// TwinCAT 3 PLC project Untitled1
// ProgramVersion: 3.1.4023.0
// libraries:
//   Tc2_HVAC, * (Beckhoff Automation GmbH)
//   Tc2_Standard, * (Beckhoff Automation GmbH)
//   Tc2_System, * (Beckhoff Automation GmbH)
//   Tc3_Module, * (Beckhoff Automation GmbH)
// project tree:
//   / PlcTask.TcTTO
//   POUs/ BARFanCoil.TcPOU, MAIN.TcPOU
//   POUs/HVAC/ AnalogInput.TcPOU, AnalogOutputEx.TcPOU, AntiBlockingDamper.TcPOU, AntiBlockingPump.TcPOU, CirculationPumpEx.TcPOU, Motor1Speed.TcPOU, Motor2Speed.TcPOU, Motor3Speed.TcPOU (not stored), OverwriteAnalog.TcPOU (not stored), Scheduler28ch.TcPOU, Scheduler7ch.TcPOU, SchedulerPublicHolidays.TcPOU, SchedulerSpecialPeriods.TcPOU (not stored), TemperatureSensorEx2.TcPOU (not stored), ThreePointActuatorMode.TcPOU, TwoPointActuatorMode.TcPOU (not stored), Work.TcPOU (not stored)
// real-time tasks:
//   TASK PlcTask: cycle T#10ms, priority 20, ADS port 350

CONFIGURATION Untitled1
    RESOURCE PLC ON TwinCAT3
        TASK PlcTask(INTERVAL := T#10ms, PRIORITY := 20);
        PROGRAM MAIN WITH PlcTask : MAIN;
    END_RESOURCE
END_CONFIGURATION

// ---- POUs/MAIN.TcPOU
PROGRAM MAIN
VAR
	
END_VAR

CirculationPumpEx();
AntiBlockingPump();
Work();
Scheduler7ch();
Scheduler28ch();
SchedulerSpecialPeriods();
SchedulerPublicHolidays();
Motor1Speed();
Motor2Speed();
Motor3Speed();
TwoPointActuatorMode();
ThreePointActuatorMode();
TemperatureSensorEx2();
OverwriteAnalog();
AnalogInput();
AnalogOutputEx();
AntiBlockingDamper();
BARFanCoil();

END_PROGRAM

// ---- POUs/HVAC/CirculationPumpEx.TcPOU
PROGRAM CirculationPumpEx
VAR
	fbHVACCirculationPumpEx: FB_HVACCirculationPumpEx;
	eDataSecurityType: E_HVACDataSecurityType := E_HVACDataSecurityType.eHVACDataSecurityType_Idle;
	bSetDefault: BOOL;
	bEnable: BOOL := TRUE;
	bExternal: BOOL;
	eCtrlModeActuator: E_HVACActuatorMode;
	rOutsideTemp: REAL;
	rValvePosition: REAL;
	bFeedbPump: BOOL := TRUE;
	bPumpProtec: BOOL := TRUE;
	bManSwitch: BOOL := TRUE;
	bCtrlVoltage: BOOL := TRUE;
	bReset: BOOL;
	bPump: BOOL;
	byState: BYTE;
	bReqExternal: BOOL;
	bReqOutsideTemp: BOOL;
	bReqValve: BOOL;
	bStateManSwitch: BOOL;
	udiSecRT_StopDelay: UDINT;
	udiSecRT_FeedbPumpDelay: UDINT;
	eStateModeActuator: Tc2_HVAC.E_HVACActuatorMode;
	bError: BOOL;
	byError: BYTE;
	bErrorPumpProtec: BOOL;
	bErrorFeedb: BOOL;
	bInvalidParameter: BOOL;
	udiSecStopDelay: UDINT;
	udiSecFeedbPumpDelay: UDINT;
	rOutsideTempHighLimit: REAL;
	rOutsideTempLowLimit: REAL;
	rValvePositionLimitOn: REAL;
	rValvePositionLimitOff: REAL;
	eReqPump: E_HVACReqPump;
END_VAR

fbHVACCirculationPumpEx(
	eDataSecurityType:=eDataSecurityType, 
	bSetDefault:=bSetDefault, 
	bEnable:=bEnable, 
	bExternal:=bExternal, 
	eCtrlModeActuator:=eCtrlModeActuator, 
	rOutsideTemp:=rOutsideTemp, 
	rValvePosition:=rValvePosition, 
	bFeedbPump:=bFeedbPump, 
	bPumpProtec:=bPumpProtec, 
	bManSwitch:=bManSwitch, 
	bCtrlVoltage:=bCtrlVoltage, 
	bReset:=bReset, 
	bPump=>bPump, 
	byState=>byState, 
	bReqExternal=>bReqExternal, 
	bReqOutsideTemp=>bReqOutsideTemp, 
	bReqValve=>bReqValve, 
	bStateManSwitch=>bStateManSwitch, 
	udiSecRT_StopDelay=>udiSecRT_StopDelay, 
	udiSecRT_FeedbPumpDelay=>udiSecRT_FeedbPumpDelay, 
	eStateModeActuator=>eStateModeActuator, 
	bError=>bError, 
	byError=>byError, 
	bErrorPumpProtec=>bErrorPumpProtec, 
	bErrorFeedb=>bErrorFeedb, 
	bInvalidParameter=>bInvalidParameter, 
	udiSecStopDelay:=udiSecStopDelay, 
	udiSecFeedbPumpDelay:=udiSecFeedbPumpDelay, 
	rOutsideTempHighLimit:=rOutsideTempHighLimit, 
	rOutsideTempLowLimit:=rOutsideTempLowLimit, 
	rValvePositionLimitOn:=rValvePositionLimitOn, 
	rValvePositionLimitOff:=rValvePositionLimitOff, 
	eReqPump:=eReqPump);

END_PROGRAM

// ---- POUs/HVAC/AntiBlockingPump.TcPOU
PROGRAM AntiBlockingPump
VAR
	fbHVACAntiBlockingPump: FB_HVACAntiBlockingPump;
	eDataSecurityType: E_HVACDataSecurityType := E_HVACDataSecurityType.eHVACDataSecurityType_Idle;
	bSetDefault: BOOL;
	bEnable: BOOL;
	bDisable: BOOL;
	bIn: BOOL;
	dtSystemTime: DATE_AND_TIME;
	bReset: BOOL;
	eAntiBlockingMode: E_HVACAntiBlockingMode;
	iHoursDowntime: INT;
	iDayWeekly: INT;
	iHour: INT;
	iMinute: INT;
	iLenghtImpulse: INT;
	bOut: BOOL;
	bOutAndAntiBlocking: BOOL;
	bQAntiBlocking: BOOL;
	bInvalidParameter: BOOL;
END_VAR

fbHVACAntiBlockingPump(
	eDataSecurityType:=eDataSecurityType, 
	bSetDefault:=bSetDefault, 
	bEnable:=bEnable, 
	bDisable:=bDisable, 
	bIn:=bIn, 
	dtSystemTime:=dtSystemTime, 
	bReset:=bReset, 
	eAntiBlockingMode:=eAntiBlockingMode, 
	iHoursDowntime:=iHoursDowntime, 
	iDayWeekly:=iDayWeekly, 
	iHour:=iHour, 
	iMinute:=iMinute, 
	iLenghtImpulse:=iLenghtImpulse, 
	bOut=>bOut, 
	bOutAndAntiBlocking=>bOutAndAntiBlocking, 
	bQAntiBlocking=>bQAntiBlocking, 
	bInvalidParameter=>bInvalidParameter);

END_PROGRAM

// ---- POUs/HVAC/Scheduler7ch.TcPOU
PROGRAM Scheduler7ch
VAR
	fbHVACScheduler7ch:FB_HVACScheduler7ch;
	eDataSecurityType:E_HVACDataSecurityType := E_HVACDataSecurityType.eHVACDataSecurityType_Idle;
	bSetDefault:BOOL;
	bEnable:BOOL;
	dtSystemTime:DT;
	uiOffsetBefore:UINT;
	bReset:BOOL;
	arrTimeChannel:ARRAY[1..7] OF ST_HVACTimeChannel;
	bOutput:BOOL;
	bEdgeOn:BOOL;
	bEdgeOff:BOOL;
	tNextOn:TIME;
	tNextOff:TIME;
	bInvalidParameter:BOOL;
END_VAR

fbHVACScheduler7ch(
	eDataSecurityType:=eDataSecurityType , 
	bSetDefault:=bSetDefault, 
	bEnable:=bEnable , 
	dtSystemTime:=dtSystemTime , 
	uiOffsetBefore:=uiOffsetBefore, 
	bReset:=bReset, 
	arrTimeChannel:=arrTimeChannel, 
	bOutput=>bOutput, 
	bEdgeOn=>bEdgeOn, 
	bEdgeOff=>bEdgeOff, 
	tNextOn=>tNextOn, 
	tNextOff=>tNextOff, 
	bInvalidParameter=>bInvalidParameter
);

END_PROGRAM

// ---- POUs/HVAC/Scheduler28ch.TcPOU
PROGRAM Scheduler28ch
VAR
	fbHVACScheduler28ch:FB_HVACScheduler28ch;
	eDataSecurityType:E_HVACDataSecurityType := E_HVACDataSecurityType.eHVACDataSecurityType_Idle;
	bSetDefault:BOOL;
	bEnable:BOOL;
	dtSystemTime:DT;
	uiOffsetBefore:UINT;
	bReset:BOOL;
	arrTimeChannel2:ARRAY[1..28] OF ST_HVACTimeChannel;
	bOutput:BOOL;
	bEdgeOn:BOOL;
	bEdgeOff:BOOL;
	tNextOn:TIME;
	tNextOff:TIME;
	bInvalidParameter:BOOL;
END_VAR

fbHVACScheduler28ch(
	eDataSecurityType:=eDataSecurityType , 
	bSetDefault:=bSetDefault, 
	bEnable:=bEnable , 
	dtSystemTime:=dtSystemTime , 
	uiOffsetBefore:=uiOffsetBefore, 
	bReset:=bReset, 
	arrTimeChannel:=arrTimeChannel2, 
	bOutput=>bOutput, 
	bEdgeOn=>bEdgeOn, 
	bEdgeOff=>bEdgeOff, 
	tNextOn=>tNextOn, 
	tNextOff=>tNextOff, 
	bInvalidParameter=>bInvalidParameter
);

END_PROGRAM

// ---- POUs/HVAC/SchedulerPublicHolidays.TcPOU
PROGRAM SchedulerPublicHolidays
VAR
	fbHVACSchedulerPublicHolidays:FB_HVACSchedulerPublicHolidays;
	eDataSecurityType:E_HVACDataSecurityType := E_HVACDataSecurityType.eHVACDataSecurityType_Idle;
	bSetDefault:BOOL;
	bEnable:BOOL;
	dtSystemTime:DT;
	bReset:BOOL;
	arrHoliday:ARRAY[1..20] OF ST_HVACHoliday;
	bOutput:BOOL;
	bEdgeOn:BOOL;
	bEdgeOff:BOOL;
	tNextOn:TIME;
	tNextOff:TIME;
	bInvalidParameter:BOOL;
END_VAR

fbHVACSchedulerPublicHolidays(
	eDataSecurityType:=eDataSecurityType , 
	bSetDefault:= bSetDefault, 
	bEnable:=bEnable, 
	dtSystemTime:=dtSystemTime, 
	bReset:=bReset, 
	arrHoliday:=arrHoliday, 
	bOutput=>bOutput, 
	bEdgeOn=>bEdgeOn, 
	bEdgeOff=>bEdgeOff, 
	tNextOn=>tNextOn, 
	tNextOff=>tNextOff, 
	bInvalidParameter=>bInvalidParameter);

END_PROGRAM

// ---- POUs/HVAC/Motor1Speed.TcPOU
PROGRAM Motor1Speed
VAR
	fbHVACMotor1Speed: FB_HVACMotor1Speed;
	eDataSecurityType: E_HVACDataSecurityType := E_HVACDataSecurityType.eHVACDataSecurityType_Idle;
	bSetDefault: BOOL;
	bEnable: BOOL;
	bAuto: BOOL;
	eCtrlModeActuator: E_HVACActuatorMode;
	bMotorProtec: BOOL;
	bFeedbContactor: BOOL;
	bFeedbProcess: BOOL;
	bRepairSwitch: BOOL;
	bManSwitch: BOOL;
	bCtrlVoltage: BOOL;
	bReset: BOOL;
	bMotor: BOOL;
	byState: BYTE;
	bStateAuto: BOOL;
	bStateRepairSwitch: BOOL;
	bStateManSwitch: BOOL;
	eStateModeActuator: Tc2_HVAC.E_HVACActuatorMode;
	bErrorGeneral: BOOL;
	byError: BYTE;
	bErrorMotorprotec: BOOL;
	bErrorFeedbContactor: BOOL;
	bErrorFeedbProcess: BOOL;
	bInvalidParameter: BOOL;
	tStartDelay: TIME;
	tStopDelay: TIME;
	tDelayFeedbContactor: TIME;
	tFeedbProcessTimer: TIME;
	tDelayFeedbProcess: TIME;
END_VAR

fbHVACMotor1Speed(
	eDataSecurityType:=eDataSecurityType, 
	bSetDefault:=bSetDefault, 
	bEnable:=bEnable, 
	bAuto:=bAuto, 
	eCtrlModeActuator:=eCtrlModeActuator, 
	bMotorProtec:=bMotorProtec, 
	bFeedbContactor:=bFeedbContactor, 
	bFeedbProcess:=bFeedbProcess, 
	bRepairSwitch:=bRepairSwitch, 
	bManSwitch:=bManSwitch, 
	bCtrlVoltage:=bCtrlVoltage, 
	bReset:=bReset, 
	bMotor=>bMotor, 
	byState=>byState, 
	bStateAuto=>bStateAuto, 
	bStateRepairSwitch=>bStateRepairSwitch, 
	bStateManSwitch=>bStateManSwitch, 
	eStateModeActuator=>eStateModeActuator, 
	bErrorGeneral=>bErrorGeneral, 
	byError=>byError, 
	bErrorMotorprotec=>bErrorMotorprotec, 
	bErrorFeedbContactor=>bErrorFeedbContactor, 
	bErrorFeedbProcess=>bErrorFeedbProcess, 
	bInvalidParameter=>bInvalidParameter, 
	tStartDelay:=tStartDelay, 
	tStopDelay:=tStopDelay, 
	tDelayFeedbContactor:=tDelayFeedbContactor, 
	tFeedbProcessTimer:=tFeedbProcessTimer, 
	tDelayFeedbProcess:=tDelayFeedbProcess);

END_PROGRAM

// ---- POUs/HVAC/Motor2Speed.TcPOU
PROGRAM Motor2Speed
VAR
	fbHVACMotor2Speed: FB_HVACMotor2Speed;
	eDataSecurityType: E_HVACDataSecurityType := E_HVACDataSecurityType.eHVACDataSecurityType_Idle;
	bSetDefault: BOOL;
	bEnable: BOOL;
	bAutoSpeed1: BOOL;
	bAutoSpeed2: BOOL;
	eCtrlModeActuator: E_HVACActuatorMode;
	bMotorProtecSpeed1: BOOL;
	bMotorProtecSpeed2: BOOL;
	bFeedbContactorSpeed1: BOOL;
	bFeedbContactorSpeed2: BOOL;
	bFeedbProcess: BOOL;
	bRepairSwitch: BOOL;
	bManSwitch: BOOL;
	bCtrlVoltage: BOOL;
	bReset: BOOL;
	bMotorSpeed1: BOOL;
	bMotorSpeed2: BOOL;
	byState: BYTE;
	bStateAutoSpeed1: BOOL;
	bStateAutoSpeed2: BOOL;
	bStateRepairSwitch: BOOL;
	bStateManSwitch: BOOL;
	eStateModeActuator: Tc2_HVAC.E_HVACActuatorMode;
	bErrorGeneral: BOOL;
	byError: BYTE;
	bErrorMotorprotecSpeed1: BOOL;
	bErrorMotorprotecSpeed2: BOOL;
	bErrorFeedbContactorSpeed1: BOOL;
	bErrorFeedbContactorSpeed2: BOOL;
	bErrorFeedbProcess: BOOL;
	bInvalidParameter: BOOL;
	tStartDelay: TIME;
	tStopDelay: TIME;
	tDelayFeedbContactorSpeed1: TIME;
	tDelayFeedbContactorSpeed2: TIME;
	tFeedbProcessTimer: TIME;
	tDelayFeedbProcess: TIME;
	tDelaySpeed1: TIME;
	tDelaySpeed1ToSpeed2: TIME;
	tDelaySpeed2ToSpeed1: TIME;
END_VAR

fbHVACMotor2Speed(
	eDataSecurityType:=eDataSecurityType, 
	bSetDefault:=bSetDefault, 
	bEnable:=bEnable, 
	bAutoSpeed1:=bAutoSpeed1, 
	bAutoSpeed2:=bAutoSpeed2, 
	eCtrlModeActuator:=eCtrlModeActuator, 
	bMotorProtecSpeed1:=bMotorProtecSpeed1, 
	bMotorProtecSpeed2:=bMotorProtecSpeed2, 
	bFeedbContactorSpeed1:=bFeedbContactorSpeed1, 
	bFeedbContactorSpeed2:=bFeedbContactorSpeed2, 
	bFeedbProcess:=bFeedbProcess, 
	bRepairSwitch:=bRepairSwitch, 
	bManSwitch:=bManSwitch, 
	bCtrlVoltage:=bCtrlVoltage, 
	bReset:=bReset, 
	bMotorSpeed1=>bMotorSpeed1, 
	bMotorSpeed2=>bMotorSpeed2, 
	byState=>byState, 
	bStateAutoSpeed1=>bStateAutoSpeed1, 
	bStateAutoSpeed2=>bStateAutoSpeed2, 
	bStateRepairSwitch=>bStateRepairSwitch, 
	bStateManSwitch=>bStateManSwitch, 
	eStateModeActuator=>eStateModeActuator, 
	bErrorGeneral=>bErrorGeneral, 
	byError=>byError, 
	bErrorMotorprotecSpeed1=>bErrorMotorprotecSpeed1, 
	bErrorMotorprotecSpeed2=>bErrorMotorprotecSpeed2, 
	bErrorFeedbContactorSpeed1=>bErrorFeedbContactorSpeed1, 
	bErrorFeedbContactorSpeed2=>bErrorFeedbContactorSpeed2, 
	bErrorFeedbProcess=>bErrorFeedbProcess, 
	bInvalidParameter=>bInvalidParameter, 
	tStartDelay:=tStartDelay, 
	tStopDelay:=tStopDelay, 
	tDelayFeedbContactorSpeed1:=tDelayFeedbContactorSpeed1, 
	tDelayFeedbContactorSpeed2:=tDelayFeedbContactorSpeed2, 
	tFeedbProcessTimer:=tFeedbProcessTimer, 
	tDelayFeedbProcess:=tDelayFeedbProcess, 
	tDelaySpeed1:=tDelaySpeed1, 
	tDelaySpeed1ToSpeed2:=tDelaySpeed1ToSpeed2,
	tDelaySpeed2ToSpeed1:=tDelaySpeed2ToSpeed1);

END_PROGRAM

// ---- POUs/HVAC/ThreePointActuatorMode.TcPOU
PROGRAM ThreePointActuatorMode
VAR
	fbHVAC3PointActuator: FB_HVAC3PointActuator;
	eDataSecurityType: E_HVACDataSecurityType := E_HVACDataSecurityType.eHVACDataSecurityType_Idle;
	bSetDefault: BOOL;
	bEnable: BOOL;
	bAutoOpen: BOOL;
	bAutoClose: BOOL;
	eCtrlModeActuator: E_HVAC3PointActuatorMode;
	bManSwitch: BOOL;
	rFeedb: REAL;
	bCtrlVoltage: BOOL;
	bReset: BOOL;
	bEnableFeedbCtrl: BOOL;
	rMinValueFeedb: REAL;
	rMaxValueFeedb: REAL := 100;
	rHysteresisFeedb: REAL;
	tStrokeTime: TIME;
	bOpen: BOOL;
	bClose: BOOL;
	byState: BYTE;
	eStateModeActuator: Tc2_HVAC.E_HVAC3PointActuatorMode;
	bErrorFeedb: BOOL;
	bInvalidParameter: BOOL;
END_VAR

fbHVAC3PointActuator(
	eDataSecurityType:=eDataSecurityType,
	bSetDefault:=bSetDefault,
	bEnable:=bEnable,
	bAutoOpen:=bAutoOpen,
	bAutoClose:=bAutoClose,
	eCtrlModeActuator:=eCtrlModeActuator,
	bManSwitch:=bManSwitch,
	rFeedb:=rFeedb,
	bCtrlVoltage:=bCtrlVoltage,
	bReset:=bReset,
	bOpen=>bOpen,
	bClose=>bClose,
	byState=>byState,
	eStateModeActuator=>eStateModeActuator,
	bErrorFeedb=>bErrorFeedb,
	bInvalidParameter=>bInvalidParameter,
	bEnableFeedbCtrl:=bEnableFeedbCtrl,
	rMinValueFeedb:=rMinValueFeedb,
	rMaxValueFeedb:=rMaxValueFeedb,
	rHysteresisFeedb:=rHysteresisFeedb,
	tStrokeTime:=tStrokeTime);

END_PROGRAM

// ---- POUs/HVAC/AnalogInput.TcPOU
PROGRAM AnalogInput
VAR
	fbHVACAnalogInput: FB_HVACAnalogInput;
	eDataSecurityType: E_HVACDataSecurityType := E_HVACDataSecurityType.eHVACDataSecurityType_Idle;
	bSetDefault: BOOL;
	iRawValue: INT;
	tTaskCycleTime: TIME;
	tCtrlCycleTime: TIME;
	bEnableLimitCtrl: BOOL;
	bCtrlVoltage: BOOL;
	bReset: BOOL;
	iHighRange: INT;
	iLowRange: INT;
	rHighRange: REAL;
	rLowRange: REAL;
	rHighLimit: REAL;
	rLowLimit: REAL;
	tFilterTime: TIME;
	rOffset: REAL;
	rPresentValue: REAL;
	byState: BYTE;
	bError: BOOL;
	eErrorCode: Tc2_HVAC.E_HVACErrorCodes;
	bErrorHighLimit: BOOL;
	bErrorLowLimit: BOOL;
	bErrorGeneral: BOOL;
	byError: BYTE;
	bInvalidParameter: BOOL;
END_VAR

fbHVACAnalogInput(
	eDataSecurityType:=eDataSecurityType, 
	bSetDefault:=bSetDefault, 
	iRawValue:=iRawValue, 
	tTaskCycleTime:=tTaskCycleTime, 
	tCtrlCycleTime:=tCtrlCycleTime, 
	bEnableLimitCtrl:=bEnableLimitCtrl, 
	bCtrlVoltage:=bCtrlVoltage, 
	bReset:=bReset, 
	rPresentValue=>rPresentValue, 
	byState=>byState, 
	bError=>bError, 
	eErrorCode=>eErrorCode, 
	bErrorHighLimit=>bErrorHighLimit, 
	bErrorLowLimit=>bErrorLowLimit, 
	bErrorGeneral=>bErrorGeneral, 
	byError=>byError, 
	bInvalidParameter=>bInvalidParameter, 
	iHighRange:=iHighRange, 
	iLowRange:=iLowRange, 
	rHighRange:=rHighRange, 
	rLowRange:=rLowRange, 
	rHighLimit:=rHighLimit, 
	rLowLimit:=rLowLimit, 
	tFilterTime:=tFilterTime, 
	rOffset:=rOffset);

END_PROGRAM

// ---- POUs/HVAC/AnalogOutputEx.TcPOU
PROGRAM AnalogOutputEx
VAR
	fbHVACAnalogOutputEx: FB_HVACAnalogOutputEx;
	eDataSecurityType: E_HVACDataSecurityType := E_HVACDataSecurityType.eHVACDataSecurityType_Idle;
	bSetDefault: BOOL;
	bEnable: BOOL;
	rSetpoint: REAL;
	bCtrlVoltage: BOOL;
	eCtrlModeAnalogOutput: E_HVACAnalogOutputMode;
	rYManual: REAL;
	rFeedb: REAL;
	bFrost: BOOL;
	bReset: BOOL;
	rX2: REAL;
	rX1: REAL;
	iY2: INT;
	iY1: INT;
	bDirection: BOOL;
	bEnableFeedbCtrl: BOOL;
	rHysteresisFeedbCtrl: REAL;
	tDelayFeedbCtrl: TIME;
	rY: REAL;
	iYTerminal: INT;
	eStateModeAnalogOutput: Tc2_HVAC.E_HVACAnalogOutputMode;
	bManualMode: BOOL;
	byState: BYTE;
	bErrorFeedb: BOOL;
	bErrorGeneral: BOOL;
	byError: BYTE;
	bInvalidParameter: BOOL;
END_VAR

fbHVACAnalogOutputEx(
	eDataSecurityType:=eDataSecurityType, 
	bSetDefault:=bSetDefault, 
	bEnable:=bEnable, 
	rSetpoint:=rSetpoint, 
	bCtrlVoltage:=bCtrlVoltage, 
	eCtrlModeAnalogOutput:=eCtrlModeAnalogOutput, 
	rYManual:=rYManual, 
	rFeedb:=rFeedb, 
	bFrost:=bFrost, 
	bReset:=bReset, 
	rY=>rY, 
	iYTerminal=>iYTerminal, 
	eStateModeAnalogOutput=>eStateModeAnalogOutput, 
	bManualMode=>bManualMode, 
	byState=>byState, 
	bErrorFeedb=>bErrorFeedb, 
	bErrorGeneral=>bErrorGeneral, 
	byError=>byError, 
	bInvalidParameter=>bInvalidParameter, 
	rX2:=rX2, 
	rX1:=rX1, 
	iY2:=iY2, 
	iY1:=iY1, 
	bDirection:=bDirection, 
	bEnableFeedbCtrl:=bEnableFeedbCtrl, 
	rHysteresisFeedbCtrl:=rHysteresisFeedbCtrl, 
	tDelayFeedbCtrl:=tDelayFeedbCtrl);

END_PROGRAM

// ---- POUs/HVAC/AntiBlockingDamper.TcPOU
PROGRAM AntiBlockingDamper
VAR
	fbHVACAntiBlockingDamper: FB_HVACAntiBlockingDamper;
	eDataSecurityType: E_HVACDataSecurityType := E_HVACDataSecurityType.eHVACDataSecurityType_Idle;
	bSetDefault: BOOL;
	bEnable: BOOL;
	bDisable: BOOL;
	ryDamper: REAL;
	dtSystemTime: DATE_AND_TIME;
	bReset: BOOL;
	eAntiBlockingMode: E_HVACAntiBlockingMode;
	iHoursDowntime: INT;
	iDayWeekly: INT;
	iHour: INT;
	iMinute: INT;
	iLenghtImpulse: INT;
	rQDamper: REAL;
	iQDamper: INT;
	bQAntiBlocking: BOOL;
	bInvalidParameter: BOOL;
END_VAR

fbHVACAntiBlockingDamper(
	eDataSecurityType:=eDataSecurityType, 
	bSetDefault:=bSetDefault, 
	bEnable:=bEnable, 
	bDisable:=bDisable, 
	ryDamper:=ryDamper, 
	dtSystemTime:=dtSystemTime, 
	bReset:=bReset, 
	eAntiBlockingMode:=eAntiBlockingMode, 
	iHoursDowntime:=iHoursDowntime, 
	iDayWeekly:=iDayWeekly, 
	iHour:=iHour, 
	iMinute:=iMinute, 
	iLenghtImpulse:=iLenghtImpulse, 
	rQDamper=>rQDamper, 
	iQDamper=>iQDamper, 
	bQAntiBlocking=>bQAntiBlocking, 
	bInvalidParameter=>bInvalidParameter);

END_PROGRAM

// ---- POUs/BARFanCoil.TcPOU
PROGRAM BARFanCoil
VAR
	fbBARFanCoil: FB_BARFanCoil;
	eDataSecurityType: E_HVACDataSecurityType := E_HVACDataSecurityType.eHVACDataSecurityType_Idle;
	bSetDefault: BOOL;
	bEnable: BOOL;
	eCtrlFct: E_BARCtrlFct;
	rSetpoint: REAL;
	rRoomTemp: REAL;
	bStageUp: BOOL;
	bStageDown: BOOL;
	iStageManual: INT;
	bReset: BOOL;
	rDeviationXW_Stage01: REAL;
	rDeviationXW_Stage02: REAL;
	rDeviationXW_Stage03: REAL;
	rHysteresisRange: REAL;
	udiSecMINPowerOnTime: UDINT;
	iFctModeFanCoil: INT;
	udiTimePeriod: UDINT;
	bStageOff: BOOL;
	bStageAuto: BOOL;
	bStage01: BOOL;
	bStage02: BOOL;
	bStage03: BOOL;
	bFanCoilActive: BOOL;
	bPresence: BOOL;
	byState: BYTE;
	byError: BYTE;
	udiSecRT_MINPowerOnTime: UDINT;
	udiRT_TimePeriod: UDINT;
	bInvalidParameter: BOOL;
END_VAR

fbBARFanCoil(
	eDataSecurityType:=eDataSecurityType, 
	bSetDefault:=bSetDefault, 
	bEnable:=bEnable, 
	eCtrlFct:=eCtrlFct, 
	rSetpoint:=rSetpoint, 
	rRoomTemp:=rRoomTemp, 
	bStageUp:=bStageUp, 
	bStageDown:=bStageDown, 
	iStageManual:=iStageManual, 
	bReset:=bReset, 
	bStageOff=>bStageOff, 
	bStageAuto=>bStageAuto, 
	bStage01=>bStage01, 
	bStage02=>bStage02, 
	bStage03=>bStage03, 
	bFanCoilActive=>bFanCoilActive, 
	bPresence=>bPresence, 
	byState=>byState, 
	byError=>byError, 
	udiSecRT_MINPowerOnTime=>udiSecRT_MINPowerOnTime, 
	udiRT_TimePeriod=>udiRT_TimePeriod, 
	bInvalidParameter=>bInvalidParameter, 
	rDeviationXW_Stage01:=rDeviationXW_Stage01, 
	rDeviationXW_Stage02:=rDeviationXW_Stage02, 
	rDeviationXW_Stage03:=rDeviationXW_Stage03, 
	rHysteresisRange:=rHysteresisRange, 
	udiSecMINPowerOnTime:=udiSecMINPowerOnTime, 
	iFctModeFanCoil:=iFctModeFanCoil, 
	udiTimePeriod:=udiTimePeriod);

END_PROGRAM
